// TIA Portal V20 export
TYPE "TypeAxisSd"
   STRUCT
      ActualEncPos : DInt;   // actual encoder position [mm/10]
      ActualPos : DInt;   // actual position [mm/10]
      LimitSwitchMin : Bool;   // limit switch min active
      LimitSwitchMax : Bool;   // limit switch max active
      Err : Bool;   // error
      ErrEnc : Bool;   // error encoder
      PosOk : Bool;   // position ok
      Plus : Bool;   // moves plus
      Minus : Bool;   // moves minus
      refRun : Bool;   // reference running
      refOk : Bool;   // reference ok
      SetCalibratePosOk : Bool;   // set calibrated position ok
   END_STRUCT;
END_TYPE
